TYPE ST_EL2574_In :
	STRUCT
		Busy			  : BIT;
		Transmit		  : BIT;
		SendAck			  : BIT;
		UpdateAck		  : BIT;
		CommandAck		  : BIT;
		CommandReject	  : BIT;
		Warning			  : BIT;
		Error			  : BIT;
		InputCycleCounter : BYTE;
	END_STRUCT
END_TYPE

(* stored: Version 1.1.0.1
   DUT ST_EL2574_In: Id {7360ced1-7e1e-4626-9ef0-ef1223882727} *)
